% RSLogix 500 project PRACTISE-20.RSS, saved by version 8.30.00.16 %
PROJECT "UNTITLED"    % processor: Bul.1763 MicroLogix 1100 Series A %

PROGRAM FILES
  LAD 2   10 rungs

DATA FILES
  O0 OUTPUT  6 elements
  I1 INPUT  12 elements
  S2 STATUS  66 elements
  B3 BINARY  1 elements
  T4 TIMER  5 elements
  C5 COUNTER  1 elements
  R6 CONTROL  1 elements
  N7 INTEGER  20 elements
  F8 FLOAT  1 elements

LADDER 2
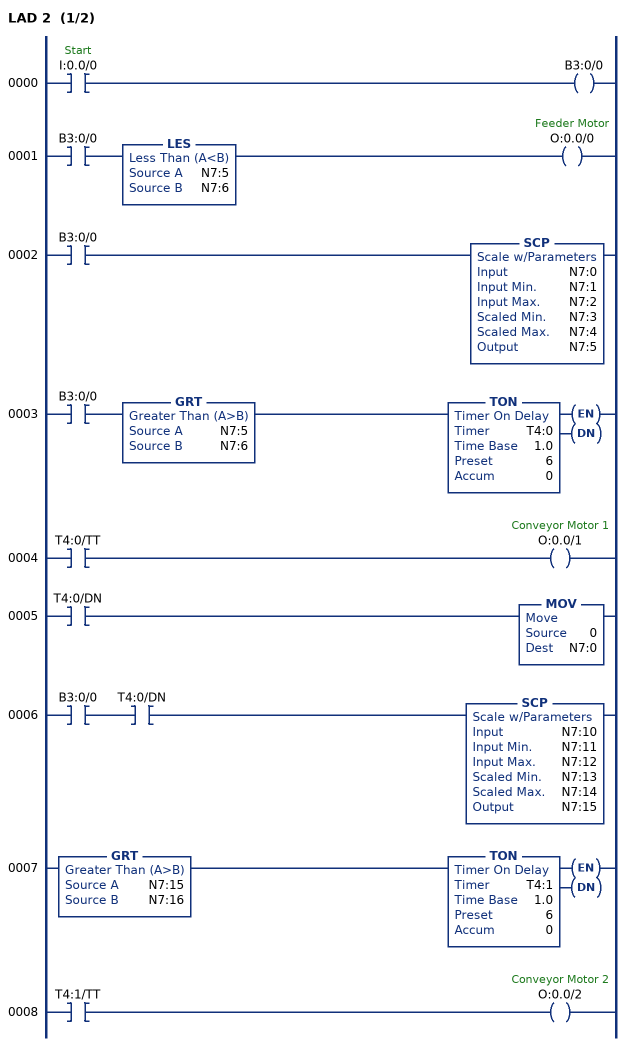
% Rung: 0 %
SOR XIC I:0.0/0 OTE B3:0/0 EOR
%   I:0.0/0  "Start" %
% Rung: 1 %
SOR XIC B3:0/0 LES N7:5 N7:6 OTE O:0.0/0 EOR
%   O:0.0/0  "Feeder Motor" %
% Rung: 2 %
SOR XIC B3:0/0 SCP N7:0 N7:1 N7:2 N7:3 N7:4 N7:5 EOR
% Rung: 3 %
SOR XIC B3:0/0 GRT N7:5 N7:6 TON T4:0 1.0 6 0 EOR
% Rung: 4 %
SOR XIC T4:0/TT OTE O:0.0/1 EOR
%   O:0.0/1  "Conveyor Motor 1" %
% Rung: 5 %
SOR XIC T4:0/DN MOV 0 N7:0 EOR
% Rung: 6 %
SOR XIC B3:0/0 XIC T4:0/DN SCP N7:10 N7:11 N7:12 N7:13 N7:14 N7:15 EOR
% Rung: 7 %
SOR GRT N7:15 N7:16 TON T4:1 1.0 6 0 EOR
% Rung: 8 %
SOR XIC T4:1/TT OTE O:0.0/2 EOR
%   O:0.0/2  "Conveyor Motor 2" %

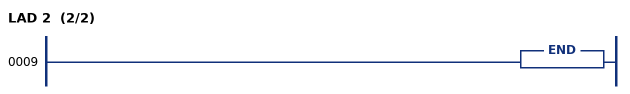
% Rung: 9 %
SOR END EOR

OTHER DOCUMENTED ADDRESSES
  I:0.0/1  "Feeder Sensor"

DATA TABLE (non-zero values as saved)
DATA T4
% .PRE .ACC %
% T4:0 % 6 0
% T4:1 % 6 0
DATA N7
% N7:0 % 10 4 20 0 50 0 10 0 0 0
% N7:10 % 10 4 20 0 50 0 10 0 0 0
